// TwinCAT 3 PLC project HeatAndSteam
// ProgramVersion: 3.1.4023.0
// libraries:
//   Tc2_DataExchange, * (Beckhoff Automation GmbH)
//   Tc2_EtherCAT, * (Beckhoff Automation GmbH)
//   Tc2_MDP, * (Beckhoff Automation GmbH)
//   Tc2_ModbusSrv, * (Beckhoff Automation GmbH)
//   Tc2_Standard, * (Beckhoff Automation GmbH)
//   Tc2_SUPS, * (Beckhoff Automation GmbH)
//   Tc2_System, * (Beckhoff Automation GmbH)
//   Tc2_Utilities, * (Beckhoff Automation GmbH)
//   Tc3_DynamicMemory, * (Beckhoff Automation GmbH)
//   Tc3_EventLogger, * (Beckhoff Automation GmbH)
//   Tc3_Module, * (Beckhoff Automation GmbH)
//   Tc3_PackML_V2, * (Beckhoff Automation GmbH)
//   Tc3_PLCopen_OpcUa, * (Beckhoff Automation GmbH)
// project tree:
//   DUTs/CELLS_INFO_STRUCTURES/Development/ DUT_STRUCT_C000000_DEV.TcDUT, DUT_STRUCT_C000001_DEV.TcDUT, DUT_STRUCT_C000002_DEV.TcDUT, DUT_STRUCT_C000003_DEV.TcDUT, DUT_STRUCT_C000004_DEV.TcDUT, DUT_STRUCT_C000005_DEV.TcDUT, DUT_STRUCT_C000006_DEV.TcDUT, DUT_STRUCT_C000007_DEV.TcDUT, DUT_STRUCT_C000008_DEV.TcDUT, DUT_STRUCT_C000009_DEV.TcDUT, DUT_STRUCT_C000010_DEV.TcDUT, DUT_STRUCT_C000012_DEV.TcDUT, DUT_STRUCT_LINECONTROLLER_DEV.TcDUT, DUT_STRUCT_TRACKSERVER_DEV.TcDUT
//   DUTs/CELLS_INFO_STRUCTURES/Production/ DUT_STRUCT_C000000_PROD.TcDUT, DUT_STRUCT_C000001_PROD.TcDUT, DUT_STRUCT_C000002_PROD.TcDUT, DUT_STRUCT_C000003_PROD.TcDUT, DUT_STRUCT_C000004_PROD.TcDUT, DUT_STRUCT_C000005_PROD.TcDUT, DUT_STRUCT_C000006_PROD.TcDUT, DUT_STRUCT_C000007_PROD.TcDUT, DUT_STRUCT_C000008_PROD.TcDUT, DUT_STRUCT_C000009_PROD.TcDUT, DUT_STRUCT_C000010_PROD.TcDUT, DUT_STRUCT_C000012_PROD.TcDUT, DUT_STRUCT_LINECONTROLLER_PROD.TcDUT, DUT_STRUCT_TRACKSERVER_PROD.TcDUT
//   ECC/Basic/ADS Comm/ E_ADS_Comm_State.TcDUT (not stored), E_ADS_Comm_Type.TcDUT (not stored), FB_ADS_Comm.TcPOU (not stored)
//   ECC/Basic/Cell/ FB_Cell_Basic.TcPOU (not stored), FB_PLC_Basic.TcPOU (not stored)
//   ECC/Basic/Common Units/ E_Units.TcDUT (not stored), FB_Units.TcPOU (not stored)
//   ECC/Basic/ GVL_BASIC.TcGVL (not stored)
//   ECC/Basic/OPC Data/ E_StationJobData.TcDUT (not stored), F_NewDeviceDataX.TcPOU (not stored), ST_InputHeader.TcDUT (not stored), ST_OutputHeaderCellInformationX.TcDUT (not stored), ST_OutputHeaderMetaInformationX.TcDUT (not stored)
//   ECC/Basic/OPC Data/Sub/ E_AlarmCategory.TcDUT (not stored), E_PML_Command.TcDUT (not stored), E_PML_Mode.TcDUT (not stored), E_PML_State.TcDUT (not stored), MaterialDataX.TcDUT (not stored), MaterialXMapping.TcDUT (not stored), ST_DataPointX.TcDUT (not stored), ST_DeviceDataX.TcDUT (not stored), ST_ErrorWarningDataX.TcDUT (not stored), ST_ManipulateMLX.TcDUT (not stored), ST_MaterialDataX.TcDUT (not stored), ST_OutputHeaderCellInformationStationInformationOperationInformationX.TcDUT (not stored), ST_OutputHeaderCellInformationStationX.TcDUT (not stored), ST_OutputHeaderTransportInformationX.TcDUT (not stored), ST_SKURestriction.TcDUT (not stored), ST_ToolDataX.TcDUT (not stored), ToolDataX.TcDUT (not stored), ToolX.TcDUT (not stored), ToolXMapping.TcDUT (not stored)
//   ECC/Basic/OPC Data/Sub/Input/ ST_InputModeState.TcDUT (not stored)
//   ECC/Basic/OPC Data/Sub/Output/ ST_Energy.TcDUT (not stored), ST_Exhaust.TcDUT (not stored), ST_Fluid.TcDUT (not stored), ST_JobDataOut.TcDUT (not stored), ST_OperationalDataOPxxxxx.TcDUT (not stored), ST_OutputErrorWarning.TcDUT (not stored), ST_OutputModeState.TcDUT (not stored), ST_OutputOEE.TcDUT (not stored)
//   ECC/Basic/Station/ FB_Station_Basic.TcPOU (not stored)
//   ECC/Basic/TrackClient/DUT/ E_CellType.TcDUT (not stored), E_MMDirection.TcTLEO (not stored), E_MMStationBuffer.TcTLEO (not stored), E_MMTrafficLightColor.TcTLEO (not stored), E_MMVehicleCommand.TcTLEO (not stored), E_MMVehicleInputType.TcTLEO (not stored), ST_MethodArgumentData.TcDUT (not stored), ST_MMBuffer.TcDUT (not stored), ST_MMLocation.TcDUT (not stored), ST_MMStation.TcDUT (not stored), ST_MMVehicleFlagData.TcDUT (not stored), ST_MMVehicleStatusData.TcDUT (not stored), ST_OPCUA_MethodData.TcDUT (not stored)
//   ECC/Basic/TrackClient/Enums/ E_CarrierStatus.TcDUT (not stored), E_MMPathMotionStatus.TcTLEO (not stored), E_MMPathState.TcTLEO (not stored), E_MMServerStatus.TcTLEO (not stored), E_OPC_UA_Errors.TcDUT (not stored), E_TrackClientState.TcDUT (not stored), E_TrackState.TcDUT (not stored), E_VehicleMoveState.TcDUT (not stored)
//   ECC/Basic/TrackClient/ E_CommandDataState.TcDUT (not stored), E_MappingDataState.TcDUT (not stored), E_ReworkDataState.TcDUT (not stored), FB_TrackClient_Basic.TcPOU (not stored)
//   ECC/Basic/TrackClient/GVLs/ GlobalConstants.TcGVL (not stored)
//   ECC/Basic/TrackClient/Method Data/Cell/ ST_GetCellIndexData.TcDUT (not stored), ST_GetCellIndexDataIn.TcDUT (not stored), ST_GetCellIndexDataOut.TcDUT (not stored)
//   ECC/Basic/TrackClient/Method Data/Data/ E_MaterialType.TcDUT (not stored), E_ToolType.TcDUT (not stored), ST_AddReservationData.TcDUT (not stored), ST_AddReservationDataIn.TcDUT (not stored), ST_AddReservationDataOut.TcDUT (not stored), ST_RemoveReservationData.TcDUT (not stored), ST_RemoveReservationDataIn.TcDUT (not stored), ST_RemoveReservationDataOut.TcDUT (not stored), ST_UpdateStationBufferData.TcDUT (not stored), ST_UpdateStationBufferDataIn.TcDUT (not stored), ST_UpdateStationBufferDataOut.TcDUT (not stored), ST_UpdateVehicleDataData.TcDUT (not stored) (excluded from build), ST_UpdateVehicleDataDataIn.TcDUT (not stored) (excluded from build), ST_UpdateVehicleDataDataOut.TcDUT (not stored) (excluded from build), ST_UpdateVehicleMappingDataData.TcDUT (not stored), ST_UpdateVehicleMappingDataDataIn.TcDUT (not stored), ST_UpdateVehicleMappingDataDataOut.TcDUT (not stored), ST_UpdateVehicleMontageData.TcDUT (not stored), ST_UpdateVehicleMontageDataIn.TcDUT (not stored), ST_UpdateVehicleMontageDataOut.TcDUT (not stored), ST_UpdateVehicleOwnerData.TcDUT (not stored), ST_UpdateVehicleOwnerDataIn.TcDUT (not stored), ST_UpdateVehicleOwnerDataOut.TcDUT (not stored), ST_UpdateVehicleReservationDataData.TcDUT (not stored), ST_UpdateVehicleReservationDataDataIn.TcDUT (not stored), ST_UpdateVehicleReservationDataDataOut.TcDUT (not stored), ST_UpdateVehicleReworkDataData.TcDUT (not stored), ST_UpdateVehicleReworkDataDataIn.TcDUT (not stored), ST_UpdateVehicleReworkDataDataOut.TcDUT (not stored)
//   ECC/Basic/TrackClient/Method Data/MoveVehicle/ ST_MoveToBufferData.TcDUT (not stored), ST_MoveToBufferDataIn.TcDUT (not stored), ST_MoveToBufferDataOut.TcDUT (not stored), ST_MoveToDecisionPointData.TcDUT (not stored), ST_MoveToDecisionPointDataIn.TcDUT (not stored), ST_MoveToDecisionPointDataOut.TcDUT (not stored), ST_MoveToPositionData.TcDUT (not stored), ST_MoveToPositionDataIn.TcDUT (not stored), ST_MoveToPositionDataOut.TcDUT (not stored), ST_MoveToScannerData.TcDUT (not stored), ST_MoveToScannerDataIn.TcDUT (not stored), ST_MoveToScannerDataOut.TcDUT (not stored), ST_MoveToStationDataIn.TcDUT (not stored), ST_MoveToStationDataOut.TcDUT (not stored), ST_MoveToStationInData.TcDUT (not stored), ST_MoveToStationOutData.TcDUT (not stored), ST_MoveVehicleStatusData.TcDUT (not stored), ST_MoveVehicleStatusDataIn.TcDUT (not stored), ST_MoveVehicleStatusDataOut.TcDUT (not stored)
//   ECC/Basic/TrackClient/Method Data/Path/ ST_AddPathData.TcDUT (not stored), ST_AddPathDataIn.TcDUT (not stored), ST_AddPathDataOut.TcDUT (not stored), ST_RemovePathData.TcDUT (not stored), ST_RemovePathDataIn.TcDUT (not stored), ST_RemovePathDataOut.TcDUT (not stored), ST_ResetPathData.TcDUT (not stored), ST_ResetPathDataIn.TcDUT (not stored), ST_ResetPathDataOut.TcDUT (not stored), ST_ResumePathData.TcDUT (not stored), ST_ResumePathDataIn.TcDUT (not stored), ST_ResumePathDataOut.TcDUT (not stored), ST_StartPathData.TcDUT (not stored), ST_StartPathDataIn.TcDUT (not stored), ST_StartPathDataOut.TcDUT (not stored), ST_SuspendPathData.TcDUT (not stored), ST_SuspendPathDataIn.TcDUT (not stored), ST_SuspendPathDataOut.TcDUT (not stored)
//   ECC/Basic/TrackClient/Method Data/Segment/ ST_AddPathSegmentData.TcDUT (not stored), ST_AddPathSegmentDataIn.TcDUT (not stored), ST_AddPathSegmentDataOut.TcDUT (not stored), ST_GetPathSegmentVehicleCountData.TcDUT (not stored), ST_GetPathSegmentVehicleCountDataIn.TcDUT (not stored), ST_GetPathSegmentVehicleCountDataOut.TcDUT (not stored), ST_RemovePathSegmentData.TcDUT (not stored), ST_RemovePathSegmentDataIn.TcDUT (not stored), ST_RemovePathSegmentDataOut.TcDUT (not stored)
//   ECC/Basic/TrackClient/Method Data/Station/ ST_AddStationData.TcDUT (not stored), ST_AddStationDataIn.TcDUT (not stored), ST_AddStationDataOut.TcDUT (not stored), ST_AddStationDoubleData.TcDUT (not stored), ST_AddStationDoubleDataIn.TcDUT (not stored), ST_AddStationDoubleDataOut.TcDUT (not stored), ST_AddStationSingleData.TcDUT (not stored), ST_AddStationSingleDataIn.TcDUT (not stored), ST_AddStationSingleDataOut.TcDUT (not stored), ST_AdjustBufferPosData.TcDUT (not stored), ST_AdjustBufferPosDataIn.TcDUT (not stored), ST_AdjustBufferPosDataOut.TcDUT (not stored), ST_EnableStationData.TcDUT (not stored), ST_EnableStationDataIn.TcDUT (not stored), ST_EnableStationDataOut.TcDUT (not stored), ST_RemoveStationData.TcDUT (not stored), ST_RemoveStationDataIn.TcDUT (not stored), ST_RemoveStationDataOut.TcDUT (not stored)
//   ECC/Basic/TrackClient/Method Data/TrafficLight/ ST_AddTrafficLightData.TcDUT (not stored), ST_AddTrafficLightDataIn.TcDUT (not stored), ST_AddTrafficLightDataOut.TcDUT (not stored), ST_RemoveTrafficLightData.TcDUT (not stored), ST_RemoveTrafficLightDataIn.TcDUT (not stored), ST_RemoveTrafficLightDataOut.TcDUT (not stored), ST_SetTrafficLightColorData.TcDUT (not stored), ST_SetTrafficLightColorDataIn.TcDUT (not stored), ST_SetTrafficLightColorDataOut.TcDUT (not stored), ST_TrafficLightColorData.TcDUT (not stored), ST_TrafficLightColorDataIn.TcDUT (not stored), ST_TrafficLightColorDataOut.TcDUT (not stored)
//   ECC/Basic/TrackClient/Node Data/ E_OPC_NodeType.TcDUT (not stored), ST_ReadCellData.TcDUT (not stored), ST_ReadNodeData.TcDUT (not stored), ST_ReadPathData.TcDUT (not stored), ST_ReadPathData_OLD.TcDUT (not stored), ST_ReadStationData.TcDUT (not stored), ST_ReadVehicleData.TcDUT (not stored), ST_ReadVehicleData_OLD.TcDUT (not stored), ST_StatusCell.TcDUT (not stored), ST_StatusNode.TcDUT (not stored), ST_StatusPath.TcDUT (not stored), ST_StatusStation.TcDUT (not stored), ST_StatusVehicle.TcDUT (not stored)
//   ECC/Basic/TrackClient/Node Data/SUB/ ST_ReservationData.TcDUT (not stored)
//   ECC/Basic/TrackClient/OPC Data/ ST_InputTransport.TcDUT (not stored), ST_OutputTransport.TcDUT (not stored)
//   ECC/Basic/TrackClient/OPC Data/Sub/ ST_BufferIndexX.TcDUT (not stored), ST_CarrierX.TcDUT (not stored), ST_InputTransportAdditionalData.TcDUT (not stored), ST_InputTransportAdditionalDataMESHandShake.TcDUT (not stored), ST_InputTransportAdditionalDataSettings.TcDUT (not stored), ST_InputTransportCommand.TcDUT (not stored), ST_InputTransportConfiguration.TcDUT (not stored), ST_InputTransportMapping.TcDUT (not stored), ST_OutputTransportAdditionalData.TcDUT (not stored), ST_OutputTransportConfiguration.TcDUT (not stored), ST_OutputTransportMapping.TcDUT (not stored), ST_OutputTransportStatus.TcDUT (not stored), ST_StationBufferStatus.TcDUT (not stored), ST_StationBufferX.TcDUT (not stored), ST_StationConfigX.TcDUT (not stored), ST_StatusBuffer.TcDUT (not stored), ST_TrackLocation.TcDUT (not stored), ST_TransportMappingCarrier.TcDUT (not stored), ST_TransportMappingStationBuffer.TcDUT (not stored)
//   ECC/Cell_Unit_4/ E_VehicleOnStation.TcDUT (not stored), FB_Cell_Unit_4.TcPOU, FB_OPC_Cell_Unit_4.TcPOU (not stored), ST_VehicleInHS.TcDUT (not stored)
//   ECC/Cell_Unit_4/HeatAndSteamDeviceDriver/ FB_EMS_HS.TcPOU (not stored), U_EMS_HS_Read.TcDUT (not stored), U_EMS_HS_Write.TcDUT (not stored)
//   ECC/Cell_Unit_4/HeatAndSteamDeviceDriver/Sub/ E_EMS_HS_Status.TcDUT (not stored), ST_EMS_HS_Alarms.TcDUT (not stored), ST_EMS_HS_Command.TcDUT (not stored), ST_EMS_HS_Read.TcDUT (not stored), ST_EMS_HS_States.TcDUT (not stored), ST_EMS_HS_Write.TcDUT (not stored)
//   ECC/Cell_Unit_4/HeatAndSteam/ FB_HeatAndSteamOUT.TcPOU (not stored), F_CalcValuesHeatSteam.TcPOU (not stored), stStationVehicleCmdOut.TcDUT (not stored), E_HSStationINSeq.TcDUT (not stored), FB_HeatAndSteamIN.TcPOU (not stored)
//   ECC/Cell_Unit_4/HeatAndSteam/OPC Data/Sub/AdditionalData/ ST_InputStationHSAdditionalDataOP11600.TcDUT (not stored), ST_InputStationHSAdditionalDataOP11601.TcDUT (not stored), ST_InputStationHSAdditionalDataMESHandShake.TcDUT (not stored), ST_InputStationHSAdditionalDataSettings.TcDUT (not stored), ST_OuputStationHSAdditionalDataOP11600.TcDUT (not stored), ST_OuputStationHSAdditionalDataOP11601.TcDUT (not stored), ST_InputStationHSAdditionalData.TcDUT (not stored), ST_InputStationHSAdditionalDataGeneral.TcDUT (not stored), ST_OutputStationHSAdditionalData.TcDUT (not stored), ST_OutputStationHSAdditionalDataGeneral.TcDUT (not stored)
//   ECC/Cell_Unit_4/HeatAndSteam/OPC Data/Sub/Configuration/ ST_InputStationHSConfigurationOP11600.TcDUT (not stored), ST_InputStationHSUpcomingConfigurationOP11601.TcDUT (not stored), ST_InputStationHSConfigurationOP11601.TcDUT (not stored), ST_OutputStationHSCurrentConfigurationOP11601.TcDUT (not stored), ST_OutputStationHSUpcomingConfigurationOP11601.TcDUT (not stored), ST_InputStationHSConfiguration.TcDUT (not stored), ST_InputStationHSConfigurationGeneral.TcDUT (not stored), ST_InputStationHSUpcomingConfiguration.TcDUT (not stored), ST_InputStationHSUpcomingConfigurationOP11600.TcDUT (not stored), ST_OutputStationHSConfigurationOP11600.TcDUT (not stored), ST_OutputStationHSCurrentConfiguration.TcDUT (not stored), ST_OutputStationHSCurrentConfigurationGeneral.TcDUT (not stored), ST_OutputStationHSCurrentConfigurationOP11600.TcDUT (not stored), ST_OutputStationHSUpcomingConfiguration.TcDUT (not stored), ST_OutputStationHSUpcomingConfigurationOP11600.TcDUT (not stored)
//   ECC/Cell_Unit_4/HeatAndSteam/OPC Data/Sub/Control/ ST_InputStationHSControlOP11601.TcDUT (not stored), ST_InputStationHSControl.TcDUT (not stored), ST_InputStationHSControlGeneral.TcDUT (not stored), ST_InputStationHSControlOP11600.TcDUT (not stored)
//   ECC/Cell_Unit_4/HeatAndSteam/OPC Data/Sub/JobData/ ST_OutputStationHSJobDataOP11600.TcDUT (not stored), ST_InputStationHSJobDataOP11601.TcDUT (not stored), ST_OutputStationHSJobDataOP11601.TcDUT (not stored), ST_InputStationHSJobData.TcDUT (not stored), ST_InputStationHSJobDataOP11600.TcDUT (not stored), ST_OutputStationHSJobData.TcDUT (not stored)
//   ECC/Cell_Unit_4/HeatAndSteam/OPC Data/Sub/OperationalData/ ST_OutputStationHSOperationalDataOP11601.TcDUT (not stored), ST_OutputStationHSOperationalData.TcDUT (not stored), ST_OutputStationHSOperationalDataGeneral.TcDUT (not stored), ST_OutputStationHSOperationalDataOP11600.TcDUT (not stored)
//   ECC/Cell_Unit_4/OPC Data/ ST_Input.TcDUT (not stored), ST_Output.TcDUT (not stored)
//   ECC/Cell_Unit_4/OPC Data/Sub/ ST_InputCell.TcDUT (not stored), ST_InputCellAdditionalData.TcDUT (not stored), ST_InputCellAdditionalDataMESHandShake.TcDUT (not stored), ST_InputCellAdditionalDataSettings.TcDUT (not stored), ST_InputCellConfiguration.TcDUT (not stored), ST_InputCellConfigurationGeneral.TcDUT (not stored), ST_InputCellControl.TcDUT (not stored), ST_InputStation.TcDUT (not stored), ST_OutputCell.TcDUT (not stored), ST_OutputCellAdditionalData.TcDUT (not stored), ST_OutputCellConfiguration.TcDUT (not stored), ST_OutputCellConfigurationGeneral.TcDUT (not stored), ST_OutputCellOperationalData.TcDUT (not stored), ST_OutputCellSustainabilityData.TcDUT (not stored), ST_OutputHeader.TcDUT (not stored), ST_OutputHeaderCellInformation.TcDUT (not stored), ST_OutputHeaderCellInformationStation.TcDUT (not stored), ST_OutputHeaderCellInformationStationInformationOperationInformation.TcDUT (not stored), ST_OutputStation.TcDUT (not stored), ST_OutputCellOperationalDataGeneral.TcDUT (not stored)
//   ECC/Cell_Unit_4/HeatAndSteam/OPC Data/ ST_InputStationStationHS.TcDUT (not stored), ST_OutputStationStationHS.TcDUT (not stored)
//   ECC/Cell_Unit_4/HeatAndSteam/OPC Data/Sub/Information/ ST_OutputHeaderCellInformationStationHS.TcDUT (not stored)
//   ECC/Cell_Unit_4/HeatAndSteam/OPC Data/Sub/Sustainability/ ST_OutputStationHSSustainabilityData.TcDUT (not stored)
//   ECC/Components/ E_ComponentErrors.TcDUT (not stored), E_Cylinder_Cmd.TcDUT (not stored), E_Cylinder_Sta.TcDUT (not stored), FB_AI.TcPOU (not stored), FB_AO.TcPOU (not stored), FB_Basic.TcPOU (not stored), FB_Blink.TcPOU (not stored), FB_Cylinder.TcPOU (not stored), FB_DI.TcPOU (not stored), FB_DO.TcPOU (not stored), FB_LIN_TRAFO.TcPOU (not stored), F_ECat_OK.TcPOU (not stored), GVL_Components.TcGVL (not stored)
//   ECC/Components/TwinSAFE/ E_TwinSAFE_Group_Diag.TcDUT (not stored), E_TwinSAFE_Group_State.TcDUT (not stored), E_TwinSAFE_Logic_State.TcDUT (not stored), FB_TwinSAFE_Group.TcPOU (not stored)
//   ECC/Tools/ E_Method.TcDUT (not stored), E_OPCUA_Client_Seq.TcDUT (not stored), FB_CheckHeartBeat.TcPOU (not stored), FB_GenerateHeartBeat.TcPOU (not stored), FB_GetCPULoad.TcPOU (not stored), FB_GetCPULoadPLC.TcPOU (not stored), FB_GetCPUTemp.TcPOU (not stored), FB_GetIPCSerial.TcPOU (not stored), FB_GetSafetyTemp.TcPOU (not stored), FB_GetTimePML.TcPOU (not stored), FB_OPCUA_Client_Basic.TcPOU (not stored), FB_OPCUA_Client_CallMethod.TcPOU (not stored), FB_OPCUA_Client_ReadVar.TcPOU (not stored), FB_OPCUA_GetRecipe.TcPOU (not stored), FB_OPCUA_ReadVar_BAK.TcPOU (not stored), F_Array_Sort.TcPOU (not stored), F_LogLine.TcPOU (not stored), F_StringCompNoCase.TcPOU (not stored), ST_OPC_Client_Data.TcDUT (not stored), ST_OutputArgInfoAndData_Basis.TcDUT (not stored), ST_Test.TcDUT (not stored)
//   ECC/Tools/LogToFile/ FB_GetFifo.TcPOU (not stored), FB_LogToFile.TcPOU (not stored), FB_SetFifo.TcPOU (not stored), F_LogFile.TcPOU (not stored), F_PadWith.TcPOU (not stored), GVL_Log.TcGVL (not stored), ST_String_FIFO.TcDUT (not stored)
//   ECC/TrackClient/Buffer Control/ FB_BufferControl.TcPOU (not stored), ST_BufferControl.TcDUT (not stored)
//   ECC/TrackClient/Enums/ E_BufferState.TcDUT (not stored), E_BufferStates.TcDUT (not stored), E_PostBufferInState.TcDUT (not stored), E_DecisionPointState.TcDUT (not stored), E_ExitPointState.TcDUT (not stored), E_StationState.TcDUT (not stored), E_PostBufferOutState.TcDUT (not stored)
//   ECC/TrackClient/ FB_TrackClient.TcPOU (not stored)
//   ECC/TrackClient/Station Control/ E_StationBufferState.TcDUT (not stored), E_StationInOutState.TcDUT (not stored), FB_StationControl.TcPOU (not stored), ST_StationControlData.TcDUT (not stored)
//   GVLs/ GVL.TcGVL
//   / PlcTask.TcTTO (not stored)
//   POUs/ MAIN.TcPOU
// real-time tasks:
//   TASK PlcTask: cycle T#10ms, priority 20, ADS port 350
// I/O:
//   DEVICE PCI (EtherCAT) (disabled), AmsNetId 10.128.16.81.2.1
//     BusCoupler (EK1200) [EK1200-5000 EtherCAT Power supply (2A E-Bus)]
//       License (EL6070-0033) [EL6070-0033 1Ch. Licence key terminal, individual licences]
//       End (EL9011) [EL9011 End Terminal]
// variable links:
//   HeatAndSteam/HeatAndSteam Instance <-> PCI (EtherCAT)/BusCoupler (EK1200)/License (EL6070-0033)
//     PlcTask Inputs/MAIN.fbUnit4.License_AdsAdrr <-> InfoData/AdsAddr
//     PlcTask Inputs/MAIN.fbUnit4.License_State <-> InfoData/State
//     PlcTask Inputs/MAIN.fbUnit4.fbSafetyTemp.sSafetyNetID/port <-> InfoData/AdsAddr/port

// ---- DUTs/CELLS_INFO_STRUCTURES/Development/DUT_STRUCT_C000000_DEV.TcDUT
TYPE DUT_STRUCT_C000000_DEV :
STRUCT
	sCellName			:STRING := 'C000000';
	sIpAddress			:STRING := '10.155.180.5';
	sAmsNetId			:STRING := '10.155.180.5.1.1';
	sOpcUaURL			:STRING := 'opc.tcp://10.155.180.5:4840';
	sUhfRfidOpcUaURL	:STRING := 'opc.tcp://10.155.180.5:4840';
	sHfRfidOpcUaURL		:STRING := 'opc.tcp://10.155.180.5:4840';
	sStation1			:STRING := 'S00000A';
END_STRUCT
END_TYPE

// ---- DUTs/CELLS_INFO_STRUCTURES/Development/DUT_STRUCT_C000001_DEV.TcDUT
TYPE DUT_STRUCT_C000001_DEV :
STRUCT
	sCellName			:STRING := 'C000001';
	sIpAddress			:STRING := '';
	sAmsNetId			:STRING := '';
	sOpcUaURL			:STRING := 'opc.tcp://:4840';
	sStation1			:STRING := 'S000008';
	sStation2			:STRING := 'S000009';
END_STRUCT
END_TYPE

// ---- DUTs/CELLS_INFO_STRUCTURES/Development/DUT_STRUCT_C000002_DEV.TcDUT
TYPE DUT_STRUCT_C000002_DEV :
STRUCT
	sCellName			:STRING := 'C000002';
	sIpAddress			:STRING := '';
	sAmsNetId			:STRING := '';
	sOpcUaURL			:STRING := 'opc.tcp://:4840';
	sStation1			:STRING := 'S000007';
END_STRUCT
END_TYPE

// ---- DUTs/CELLS_INFO_STRUCTURES/Development/DUT_STRUCT_C000003_DEV.TcDUT
TYPE DUT_STRUCT_C000003_DEV :
STRUCT
	sCellName			:STRING := 'C000003';
	sIpAddress			:STRING := '';
	sAmsNetId			:STRING := '';
	sOpcUaURL			:STRING := 'opc.tcp://:4840';
	sStation1			:STRING := 'S000006';
END_STRUCT
END_TYPE

// ---- DUTs/CELLS_INFO_STRUCTURES/Development/DUT_STRUCT_C000004_DEV.TcDUT
TYPE DUT_STRUCT_C000004_DEV :
STRUCT
	sCellName			:STRING := 'C000004';
	sIpAddress			:STRING := '10.155.180.12';
	sAmsNetId			:STRING := '10.155.180.12.1.1';
	sOpcUaURL			:STRING := 'opc.tcp://10.155.180.12:4840';
	sStation1			:STRING := 'S000003';
END_STRUCT
END_TYPE

// ---- DUTs/CELLS_INFO_STRUCTURES/Development/DUT_STRUCT_C000005_DEV.TcDUT
TYPE DUT_STRUCT_C000005_DEV :
STRUCT
	sCellName			:STRING := 'C000005';
	sIpAddress			:STRING := '';
	sAmsNetId			:STRING := '';
	sOpcUaURL			:STRING := 'opc.tcp://:4840';
	sStation1			:STRING := 'S000001';
END_STRUCT
END_TYPE

// ---- DUTs/CELLS_INFO_STRUCTURES/Development/DUT_STRUCT_C000006_DEV.TcDUT
TYPE DUT_STRUCT_C000006_DEV :
STRUCT
	sCellName			:STRING := 'C000006';
	sIpAddress			:STRING := '';
	sAmsNetId			:STRING := '';
	sOpcUaURL			:STRING := 'opc.tcp://:4840';
	sStation1			:STRING := 'S000002';
END_STRUCT
END_TYPE

// ---- DUTs/CELLS_INFO_STRUCTURES/Development/DUT_STRUCT_C000007_DEV.TcDUT
TYPE DUT_STRUCT_C000007_DEV :
STRUCT
	sCellName			:STRING := 'C0000007';
	sIpAddress			:STRING := '';
	sAmsNetId			:STRING := '';
	sOpcUaURL			:STRING := 'opc.tcp://:4840';
	sStation1			:STRING := 'S00000B';
END_STRUCT
END_TYPE

// ---- DUTs/CELLS_INFO_STRUCTURES/Development/DUT_STRUCT_C000008_DEV.TcDUT
TYPE DUT_STRUCT_C000008_DEV :
STRUCT
	sCellName			:STRING := 'C000008';
	sIpAddress			:STRING := '';
	sAmsNetId			:STRING := '';
	sOpcUaURL			:STRING := 'opc.tcp://:4840';
	sStation1			:STRING := 'S000005';
END_STRUCT
END_TYPE

// ---- DUTs/CELLS_INFO_STRUCTURES/Development/DUT_STRUCT_C000009_DEV.TcDUT
TYPE DUT_STRUCT_C000009_DEV :
STRUCT
	sCellName			:STRING := 'C000009';
	sIpAddress			:STRING := '';
	sAmsNetId			:STRING := '';
	sOpcUaURL			:STRING := 'opc.tcp://:4840';
	sUhfRfidOpcUaURL	:STRING := 'opc.tcp://:4840';
	sHfRfidOpcUaURL		:STRING := 'server:opc.tcp://:4840';
	sStation1			:STRING := 'S000004';
	sLastingPC			:STRING := '';
END_STRUCT
END_TYPE

// ---- DUTs/CELLS_INFO_STRUCTURES/Development/DUT_STRUCT_C000010_DEV.TcDUT
TYPE DUT_STRUCT_C000010_DEV :
STRUCT
	sCellName			:STRING := 'C000010';
	sIpAddress			:STRING := '';
	sAmsNetId			:STRING := '';
	sOpcUaURL			:STRING := 'opc.tcp://:4840';
	sStation1			:STRING := 'S00005D';
	sStation2			:STRING := 'S00005A';
END_STRUCT
END_TYPE

// ---- DUTs/CELLS_INFO_STRUCTURES/Development/DUT_STRUCT_C000012_DEV.TcDUT
TYPE DUT_STRUCT_C000012_DEV :
STRUCT
	sCellName			:STRING := 'C000012';
	sIpAddress			:STRING := '';
	sAmsNetId			:STRING := '';
	sOpcUaURL			:STRING := 'opc.tcp://:4840';
	sStation1			:STRING := 'S000010';
END_STRUCT
END_TYPE

// ---- DUTs/CELLS_INFO_STRUCTURES/Development/DUT_STRUCT_LINECONTROLLER_DEV.TcDUT
TYPE DUT_STRUCT_LINECONTROLLER_DEV :
STRUCT
	sCellName			:STRING := 'LINECONTROLLER';
	sIpAddress			:STRING := '10.155.180.8';
	sAmsNetId			:STRING := '';
END_STRUCT
END_TYPE

// ---- DUTs/CELLS_INFO_STRUCTURES/Development/DUT_STRUCT_TRACKSERVER_DEV.TcDUT
TYPE DUT_STRUCT_TRACKSERVER_DEV :
STRUCT
	sCellName			:STRING := 'TRACKSERVER';
	sIpAddress			:STRING := '10.155.180.10';
	sAmsNetId			:STRING := '10.155.180.10.1.1';
END_STRUCT
END_TYPE

// ---- DUTs/CELLS_INFO_STRUCTURES/Production/DUT_STRUCT_C000000_PROD.TcDUT
TYPE DUT_STRUCT_C000000_PROD :
STRUCT
	sCellName			:STRING := 'C000000';
	sIpAddress			:STRING := '10.38.190.130';
	sAmsNetId			:STRING := '10.38.190.130.1.1';
	sOpcUaURL			:STRING := 'opc.tcp://10.38.190.130:4840';
	sUhfRfidOpcUaURL	:STRING := 'opc.tcp://10.38.190.132:4840';
	sHfRfidOpcUaURL		:STRING := 'opc.tcp://10.38.190.134:4840';
	sStation1			:STRING := 'S00000A';
END_STRUCT
END_TYPE

// ---- DUTs/CELLS_INFO_STRUCTURES/Production/DUT_STRUCT_C000001_PROD.TcDUT
TYPE DUT_STRUCT_C000001_PROD :
STRUCT
	sCellName			:STRING := 'C000001';
	sIpAddress			:STRING := '10.38.191.0';
	sAmsNetId			:STRING := '10.38.191.0.1.1';
	sOpcUaURL			:STRING := 'opc.tcp://10.38.191.0:4840';
	sStation1			:STRING := 'S000008';
	sStation2			:STRING := 'S000009';
END_STRUCT
END_TYPE

// ---- DUTs/CELLS_INFO_STRUCTURES/Production/DUT_STRUCT_C000002_PROD.TcDUT
TYPE DUT_STRUCT_C000002_PROD :
STRUCT
	sCellName			:STRING := 'C000002';
	sIpAddress			:STRING := '10.38.191.20';
	sAmsNetId			:STRING := '10.38.191.20.1.1';
	sOpcUaURL			:STRING := 'opc.tcp://10.38.191.20:4840';
	sStation1			:STRING := 'S000007';
END_STRUCT
END_TYPE

// ---- DUTs/CELLS_INFO_STRUCTURES/Production/DUT_STRUCT_C000003_PROD.TcDUT
TYPE DUT_STRUCT_C000003_PROD :
STRUCT
	sCellName			:STRING := 'C000003';
	sIpAddress			:STRING := '10.38.191.40';
	sAmsNetId			:STRING := '10.38.191.40.1.1';
	sOpcUaURL			:STRING := 'opc.tcp://10.38.191.40:4840';
	sStation1			:STRING := 'S000006';
END_STRUCT
END_TYPE

// ---- DUTs/CELLS_INFO_STRUCTURES/Production/DUT_STRUCT_C000004_PROD.TcDUT
TYPE DUT_STRUCT_C000004_PROD :
STRUCT
	sCellName			:STRING := 'C000004';
	sIpAddress			:STRING := '10.38.190.201';
	sAmsNetId			:STRING := '10.38.190.201.1.1';
	sOpcUaURL			:STRING := 'opc.tcp://10.38.190.201:4840';
	sStation1			:STRING := 'S000003';
END_STRUCT
END_TYPE

// ---- DUTs/CELLS_INFO_STRUCTURES/Production/DUT_STRUCT_C000005_PROD.TcDUT
TYPE DUT_STRUCT_C000005_PROD :
STRUCT
	sCellName			:STRING := 'C000005';
	sIpAddress			:STRING := '10.38.190.204';
	sAmsNetId			:STRING := '10.38.190.204.1.1';
	sOpcUaURL			:STRING := 'opc.tcp://10.38.190.204:4840';
	sStation1			:STRING := 'S000001';
END_STRUCT
END_TYPE

// ---- DUTs/CELLS_INFO_STRUCTURES/Production/DUT_STRUCT_C000006_PROD.TcDUT
TYPE DUT_STRUCT_C000006_PROD :
STRUCT
	sCellName			:STRING := 'C000006';
	sIpAddress			:STRING := '10.38.190.200';
	sAmsNetId			:STRING := '10.38.190.200.1.1';
	sOpcUaURL			:STRING := 'opc.tcp://10.38.190.200:4840';
	sStation1			:STRING := 'S000002';
END_STRUCT
END_TYPE

// ---- DUTs/CELLS_INFO_STRUCTURES/Production/DUT_STRUCT_C000007_PROD.TcDUT
TYPE DUT_STRUCT_C000007_PROD :
STRUCT
	sCellName			:STRING := 'C0000007';
	sIpAddress			:STRING := '10.38.190.203';
	sAmsNetId			:STRING := '10.38.190.203.1.1';
	sOpcUaURL			:STRING := 'opc.tcp://10.38.190.203:4840';
	sStation1			:STRING := 'S00000B';
END_STRUCT
END_TYPE

// ---- DUTs/CELLS_INFO_STRUCTURES/Production/DUT_STRUCT_C000008_PROD.TcDUT
TYPE DUT_STRUCT_C000008_PROD :
STRUCT
	sCellName			:STRING := 'C000008';
	sIpAddress			:STRING := '10.38.190.202';
	sAmsNetId			:STRING := '10.38.190.202.1.1';
	sOpcUaURL			:STRING := 'opc.tcp://10.38.190.202:4840';
	sStation1			:STRING := 'S000005';
END_STRUCT
END_TYPE

// ---- DUTs/CELLS_INFO_STRUCTURES/Production/DUT_STRUCT_C000009_PROD.TcDUT
TYPE DUT_STRUCT_C000009_PROD :
STRUCT
	sCellName			:STRING := 'C000009';
	sIpAddress			:STRING := '10.38.191.60';
	sAmsNetId			:STRING := '10.38.191.60.1.1';
	sOpcUaURL			:STRING := 'opc.tcp://10.38.191.60:4840';
	sUhfRfidOpcUaURL	:STRING := 'opc.tcp://10.38.190.132:4840';
	sHfRfidOpcUaURL		:STRING := 'server:opc.tcp://10.38.191.66:4840';
	sStation1			:STRING := 'S000004';
	sLastingPC			:STRING := '10.38.191.65';
END_STRUCT
END_TYPE

// ---- DUTs/CELLS_INFO_STRUCTURES/Production/DUT_STRUCT_C000010_PROD.TcDUT
TYPE DUT_STRUCT_C000010_PROD :
STRUCT
	sCellName			:STRING := 'C000010';
	sIpAddress			:STRING := '10.38.191.100';
	sAmsNetId			:STRING := '10.38.191.100.1.1';
	sOpcUaURL			:STRING := 'opc.tcp://10.38.191.100:4840';
	sStation1			:STRING := 'S00005D';
	sStation2			:STRING := 'S00005A';
END_STRUCT
END_TYPE

// ---- DUTs/CELLS_INFO_STRUCTURES/Production/DUT_STRUCT_C000012_PROD.TcDUT
TYPE DUT_STRUCT_C000012_PROD :
STRUCT
	sCellName			:STRING := 'C000012';
	sIpAddress			:STRING := '10.38.191.140';
	sAmsNetId			:STRING := '10.38.191.140.1.1';
	sOpcUaURL			:STRING := 'opc.tcp://10.38.191.140:4840';
	sStation1			:STRING := 'S000010';
END_STRUCT
END_TYPE

// ---- DUTs/CELLS_INFO_STRUCTURES/Production/DUT_STRUCT_LINECONTROLLER_PROD.TcDUT
TYPE DUT_STRUCT_LINECONTROLLER_PROD :
STRUCT
	sCellName			:STRING := 'LINECONTROLLER';
	sIpAddress			:STRING := '10.38.190.120';
	sAmsNetId			:STRING := '';
END_STRUCT
END_TYPE

// ---- DUTs/CELLS_INFO_STRUCTURES/Production/DUT_STRUCT_TRACKSERVER_PROD.TcDUT
TYPE DUT_STRUCT_TRACKSERVER_PROD :
STRUCT
	sCellName			:STRING := 'TRACKSERVER';
	sIpAddress			:STRING := '10.38.190.121';
	sAmsNetId			:STRING := '10.38.190.121.1.1';
END_STRUCT
END_TYPE

// ---- GVLs/GVL.TcGVL
VAR_GLOBAL CONSTANT
	{attribute 'OPC.UA.DA':='1'}
	{attribute 'OPC.UA.DA.Access' := '1'}
	{attribute 'OPC.UA.DA.Description' := 'SW Version'}
	sSWVersion			: STRING := '0.1';

	iNoOfRecipeData		: UINT := 100;
END_VAR
VAR_GLOBAL
	bLogToOutputWindow	: BOOL;		// if TRUE it will log all logs to file AND to output window
	
	// cells info for PRODUCTION
	C000000_PROD				:DUT_STRUCT_C000000_PROD;
	C000001_PROD				:DUT_STRUCT_C000001_PROD;
	C000002_PROD				:DUT_STRUCT_C000002_PROD;
	C000003_PROD				:DUT_STRUCT_C000003_PROD;
	C000004_PROD				:DUT_STRUCT_C000004_PROD;
	C000005_PROD				:DUT_STRUCT_C000005_PROD;
	C000006_PROD				:DUT_STRUCT_C000006_PROD;
	C000007_PROD				:DUT_STRUCT_C000007_PROD;
	C000008_PROD				:DUT_STRUCT_C000008_PROD;
	C000009_PROD				:DUT_STRUCT_C000009_PROD;
	C000010_PROD				:DUT_STRUCT_C000010_PROD;
	C000012_PROD				:DUT_STRUCT_C000012_PROD;
	TrackServer_PROD			:DUT_STRUCT_TRACKSERVER_PROD;
	LineController_PROD			:DUT_STRUCT_LINECONTROLLER_PROD;
	
	// cells info for DEVELOPMENT
	C000000_DEV					:DUT_STRUCT_C000000_DEV;
	C000001_DEV					:DUT_STRUCT_C000001_DEV;
	C000002_DEV					:DUT_STRUCT_C000002_DEV;
	C000003_DEV					:DUT_STRUCT_C000003_DEV;
	C000004_DEV					:DUT_STRUCT_C000004_DEV;
	C000005_DEV					:DUT_STRUCT_C000005_DEV;
	C000006_DEV					:DUT_STRUCT_C000006_DEV;
	C000007_DEV					:DUT_STRUCT_C000007_DEV;
	C000008_DEV					:DUT_STRUCT_C000008_DEV;
	C000009_DEV					:DUT_STRUCT_C000009_DEV;
	C000010_DEV					:DUT_STRUCT_C000010_DEV;
	C000012_DEV					:DUT_STRUCT_C000012_DEV;
	TrackServer_DEV				:DUT_STRUCT_TRACKSERVER_DEV;
	LineController_DEV			:DUT_STRUCT_LINECONTROLLER_DEV;
END_VAR

// ---- ECC/Cell_Unit_4/FB_Cell_Unit_4.TcPOU
FUNCTION_BLOCK FB_Cell_Unit_4 EXTENDS FB_Cell_Basic
VAR_INPUT
END_VAR
VAR_OUTPUT
	bError						: BOOL;
	iErrorID					: BOOL;
END_VAR
VAR_IN_OUT
	// Bridge data
	Input						: ST_Input;
	Output						: ST_Output;
END_VAR
VAR
// Local vars
	eSeq						: E_VehicleOnStation;
	tonSeqTimer					: TON;
	aVehiclesStationFIFO		: ARRAY[1..10] OF ST_VehicleInHS;
	aDummyVehicleStationData	: ST_VehicleInHS;
	fDistanceStation2Station	: REAL; //Distance between stations

	stDeviceInfo				: ST_DeviceIdentification;			// Device information such as serial no.
	stVehicleDataOnStation		: ST_ReadVehicleData;
	nPLCVersion					: UINT:=0;
	nScannerInterfaceVersion	: UINT:=0;	
	bInitDone					: BOOL;
	bVehicleEnterStationOS	 	: BOOL;
	bVehicleMoveToStation		: BOOL;
	iRes						: INT;
	diFifoLogTimer				: UINT;
	diVehiclesInDevice			: UINT;
	
	tonVehicleDataRead			: TON;	// To trig reading of data for vehicles in the FIFO buffer

// FunctionBlocks:
	fbStationINHeatAndSteam		: FB_HeatAndSteamIN;
	fbStationOUTHeatAndSteam	: FB_HeatAndSteamOUT;
	fbTrack						: FB_TrackClient;
	
// Start op procedure
	bBypassTrack	:	BOOL;
	nCheckValid		:	UINT;
	nIndx			:	UINT;
	nIndxStart		:	UINT;
	nIndxDone		:	UINT;
	fVel			:	REAL;
	fAcc			:	REAL;
	bStartupPrd		:	BOOL;
	
// Error / Warnings
	iST1ErrWarDataChange	: UINT;
	iST2ErrWarDataChange	: UINT;
	iTCErrWarDataChange		: UINT;
END_VAR

SUPER^(	stModeStateIn := Input.Cell.ModeState,
		stModeStateOut := Output.Cell.ModeState,
		stOEE := Output.Cell.OEE,
		stErrorWarning := Output.Cell.ErrorWarning);

// Init FB's
M_Init();

// Run components
M_Components();
		
// Device controller
M_Device_Sequence();

// Error and warnings
M_ErrorWarning();

//Sustainability Data
M_SustainabilityDataHandling();

//Clear all ticket data
IF Input.Cell.AdditionalData.ClearAll THEN
	Input.Cell.AdditionalData.ClearAll R= M_ClearAll();
END_IF

// Update PackML state/modes variables from local values
bEStopOK := TRUE;
bStartLocal;
bStopLocal;
bClearLocal;
bResetLocal := ((eCurrentState = E_PMLState.ePMLState_Complete) AND (eCommand = E_PMLCommand.ePMLCommand_Undefined)); // Automatic back to Idle when finished
bHoldLocal;
bProductionLocal;
bManualLocal;

{attribute 'object_name' := 'M_Aborted'}
METHOD M_Aborted
END_METHOD

{attribute 'object_name' := 'M_Aborting'}
METHOD M_Aborting
// Stop all moving parts


// Abort is handled internally in Brushing Station FB, follows Cell unit state!
//IF (fbScanner1.stModeStateOut.CurrentMode = E_PML_State.Aborted) THEN
//	M_StateComplete();	
//END_IF


// No moving parts, go straight to nest state
//eCommand := E_PML_Command.Undefined;
M_StateComplete();
END_METHOD

METHOD PROTECTED M_CarrierFinishInfeedToTrack : BOOL
VAR_INPUT
END_VAR

// TODO!!!
M_CarrierFinishInfeedToTrack := TRUE;
END_METHOD

METHOD PROTECTED M_CarrierFinishOutfeedToTrack : BOOL
VAR_INPUT
END_VAR

// TODO!!!
M_CarrierFinishOutfeedToTrack := TRUE;
END_METHOD

METHOD PROTECTED M_CarrierReadyInfeedFromTrack : BOOL
VAR_INPUT
END_VAR

// TODO!!!
M_CarrierReadyInfeedFromTrack := FALSE;
END_METHOD

METHOD PROTECTED M_CarrierReadyOutfeedFromTrack : BOOL
VAR_INPUT
END_VAR

// TODO!!!
M_CarrierReadyOutfeedFromTrack := TRUE;
END_METHOD

METHOD M_ClearAll : BOOL
VAR_INPUT
END_VAR
VAR
	i : USINT;
END_VAR
//Clear all ticket data on cell from OPC command

//Clear Station(s) and TrackClient
IF fbStationINHeatAndSteam.M_ClearAll() AND fbStationOUTHeatAndSteam.M_ClearAll() THEN
	M_ClearAll := fbTrack.M_ClearAll();
END_IF
	
//Clear Cell
IF M_ClearAll THEN
	 eSeq := E_VehicleOnStation.Idle;
	 
	 //Clean out FIFO
	FOR i := 1 TO 9 DO
		aVehiclesStationFIFO[i] := aDummyVehicleStationData;
	END_FOR	
	F_Logfile('Cell - All data cleared!');
END_IF
END_METHOD

{attribute 'object_name' := 'M_Clearing'}
METHOD M_Clearing
// Reset safety system

//fbScanner1.nCellStateCmd := E_PML_Command.Clear;

//fbTrack.bReset := TRUE;

//IF ((fbScanner1.stModeStateOut.CurrentMode = E_PML_State.idle) OR (fbScanner1.stModeStateOut.CurrentMode = E_PML_State.stopped)) THEN
//	M_StateComplete();
	
//	fbTrack.bReset := FALSE;
//END_IF
//eCommand := E_PML_Command.Undefined;
M_StateComplete();
END_METHOD

{attribute 'object_name' := 'M_Complete'}
METHOD M_Complete
END_METHOD

{attribute 'object_name' := 'M_Completing'}
METHOD M_Completing

VAR
	sLowHighUpperID : STRING;	
	iRes			: INT;
END_VAR

//eCommand := E_PML_Command.Undefined;
M_StateComplete();
END_METHOD

METHOD PROTECTED M_Components : BOOL
VAR_INPUT
END_VAR
VAR
END_VAR
// Run component blocks
END_METHOD

METHOD M_Device_Sequence
VAR_INPUT
END_VAR
VAR
	i			: UINT;
	iRes		: INT;
	bMoveToNext	: BOOL;
END_VAR
// Heart beat
iHeartBeatFromMES := Input.Header.HeartBeat;
Output.Header.HeartBeat := iHeartBeatToMES;

// Run Station(s) (define when each needs to run)
fbStationINHeatAndSteam(
	aVehiclesStationFIFO:= aVehiclesStationFIFO,
	stReservation:= fbTrack.P_stReservation,
	stModeStateIn:= Input.Station.Station1.ModeState, 
	stModeStateOut := Output.Station.Station1.ModeState,
	bVehicleReadyAtInput:= eSeq <> E_VehicleOnStation.Idle, 
	bVehicleReadyAtOutput:= , 
	nCellStateCmd:= DINT_TO_UINT(eCommand),
	stJobDataIn:= Input.Station.Station1.JobData,  
	stConfigIn:= Input.Station.Station1.CurrentConfiguration, 
	stUpcomingConfigIn:= Input.Station.Station1.UpcomingConfiguration, 
	stControlIn := Input.Station.Station1.Control,
	stAdditionalDataIn := Input.Station.Station1.AdditionalData,
	sDistanceInDevice := Input.Transport.Configuration.Stations[2].StationLocation1.Position - Input.Transport.Configuration.Stations[1].StationLocation1.Position,
	stVehicleDataStaion := fbTrack.P_stVehicleDataOnStation,
	stJobDataOut := Output.Station.Station1.JobData,  
	stOEE := Output.Station.Station1.OEE, 
	stErrorWarning := Output.Station.Station1.ErrorWarning, 
	stConfigOut := Output.Station.Station1.CurrentConfiguration,
	stUpcomingConfigOut := Output.Station.Station1.UpcomingConfiguration,
	stOperationalDataOut := Output.Station.Station1.OperationalData, 
	stSustainabilityData := Output.Station.Station1.SustainabilityData, 
	stAdditionalDataOut := Output.Station.Station1.AdditionalData 	);
	
fbStationOUTHeatAndSteam(
	stModeStateIn:= Input.Station.Station2.ModeState, 
	stModeStateOut := Output.Station.Station2.ModeState,
	bVehicleReadyAtInput:= , 
	bVehicleReadyAtOutput:= , 
	nCellStateCmd:= DINT_TO_UINT(eCommand),
	stJobDataIn:= Input.Station.Station2.JobData,  
	stConfigIn:= Input.Station.Station2.CurrentConfiguration, 
	stUpcomingConfigIn:= Input.Station.Station2.UpcomingConfiguration, 
	stControlIn := Input.Station.Station2.Control,
	stAdditionalDataIn := Input.Station.Station1.AdditionalData,
	stJobDataOut := Output.Station.Station2.JobData,  
	stOEE := Output.Station.Station2.OEE, 
	stErrorWarning := Output.Station.Station2.ErrorWarning, 
	stConfigOut := Output.Station.Station2.CurrentConfiguration,
	stUpcomingConfigOut := Output.Station.Station2.UpcomingConfiguration,
	stOperationalDataOut := Output.Station.Station2.OperationalData, 
	stSustainabilityData := Output.Station.Station2.SustainabilityData, 
	stAdditionalDataOut := Output.Station.Station2.AdditionalData 	);

	
// Run Track Client
fbTrack(bEnable := , // Enabled in State Resetting
		bEStopOK := TRUE,
		bSuspend := , 
		bReset:= , 
		stCommand:= Input.Transport.Command,
		stMappingIn:= input.Transport.Mapping,
		stAdditionalDataIn:= Input.Transport.AdditionalData,
		bConnectedMethod=> , 
		bBusyMethod=> , 
		bConnectedNode=> , 
		bErrorMethod=> , 
		nErrorMethodID=> , 
		bErrorNode=> , 
		nErrorNodeID=> , 
		stStatus := Output.Transport.Status,
		stMappingOut := Output.Transport.Mapping, 
		stAdditionaldataOut := Output.Transport.AdditionalData,
		bStarted=> , 
		bSuspended=> 	);


//Set Station ready for vehicle to track
fbTrack.P_StationEmptyReady := eSeq = E_VehicleOnStation.Idle;
//fbTrack.P_bStationReady:=fbStationINHeatAndSteam.bStationReadyIn;

//Vehicles on station FIFO handling
M_VehicleOnStation(iCarrierCount=>diVehiclesInDevice);


//Set station empty for track - for vehicles going straight through
fbTrack.P_bStationEmpty:= diVehiclesInDevice = 0;

//Set FIFO for Station IN and Track Client
//fbStationINHeatAndSteam.P_CarriersFIFO := aVehiclesStationFIFO;
fbTrack.P_CarriersFIFO := aVehiclesStationFIFO;
END_METHOD

METHOD PROTECTED M_ErrorWarning
VAR_INPUT
END_VAR
VAR
	iAlNo				: UINT;
	iNoOfAlarms			: UINT;
	iNoOfWarnings		: UINT;
	bST1ErrWarDataChange: BOOL;
	bST2ErrWarDataChange: BOOL;
	bCellDataChange		: BOOL;
	bTCErrWarDataChange	: BOOL;
END_VAR
//Alarm / Warnings Cell
//bCellDataChange S= 
//M_ErrorWarningObj(arErrorWaringData:= arErrorWarningDataCell,
//	bActive:= eLineCtrl_EStop <> E_TwinSAFE_Logic_State.RUN, 
//	iErrorWarningType:= 2, 
//	diErrorWarningID:= E_AlarmCategory.Safety + 0, 
//	sDeviceID:= 'Global Safety',
//	iSeverity:= 2, 
//	iNativeID:= 0, 
//	sNativeMessage:= 'Emergency stop Line Controller');

//bCellDataChange S= 
//M_ErrorWarningObj(arErrorWaringData:= arErrorWarningDataCell,
//	bActive:= NOT bEStop_OK, 
//	iErrorWarningType:= 2, 
//	diErrorWarningID:= E_AlarmCategory.Safety + 20, 
//	sDeviceID:= 'Local Safety',
//	iSeverity:= 2, 
//	iNativeID:= 0, 
//	sNativeMessage:= 'Emergency stop Cell');

//bCellDataChange S= 
//M_ErrorWarningObj(arErrorWaringData:= arErrorWarningDataCell,
//	bActive:= eSHL_F70 <> E_TwinSAFE_Logic_State.RUN, 
//	iErrorWarningType:= 2, 
//	diErrorWarningID:= E_AlarmCategory.Safety + 21, 
//	sDeviceID:= 'Local Safety',
//	iSeverity:= 2, 
//	iNativeID:= 0, 
//	sNativeMessage:= 'Emergency stop Robot');
	
//bCellDataChange S= 
//M_ErrorWarningObj(arErrorWaringData:= arErrorWarningDataCell,
//	bActive:= NOT bDoor_OK, 
//	iErrorWarningType:= 2, 
//	diErrorWarningID:= E_AlarmCategory.Safety + 22, 
//	sDeviceID:= 'Local Safety',
//	iSeverity:= 2, 
//	iNativeID:= 0, 
//	sNativeMessage:= 'Cell Door 1 Not OK');
	
//bCellDataChange S= 
//M_ErrorWarningObj(arErrorWaringData:= arErrorWarningDataCell,
//	bActive:= stStatusData.e03_11_AK01_M3011 = E_Cylinder_Sta.Cyl_Sta_Err, 
//	iErrorWarningType:= 2, 
//	diErrorWarningID:= E_AlarmCategory.LifterStation1Device + 0, 
//	sDeviceID:= 'Lifter Station 1',
//	iSeverity:= 2, 
//	iNativeID:= 0, 
//	sNativeMessage:= 'Error Radial Gripper');
	
//bCellDataChange S= 
//M_ErrorWarningObj(arErrorWaringData:= arErrorWarningDataCell,
//	bActive:= stStatusData.e03_11_AK01_M3015 = E_Cylinder_Sta.Cyl_Sta_Err, 
//	iErrorWarningType:= 2, 
//	diErrorWarningID:= E_AlarmCategory.LifterStation1Device + 1, 
//	sDeviceID:= 'Lifter Station 1',
//	iSeverity:= 2, 
//	iNativeID:= 0, 
//	sNativeMessage:= 'Error Lifter Cylinder');
	
//bCellDataChange S= 
//M_ErrorWarningObj(arErrorWaringData:= arErrorWarningDataCell,
//	bActive:= stStatusData.e03_11_AK01_M3111 = E_Cylinder_Sta.Cyl_Sta_Err, 
//	iErrorWarningType:= 2, 
//	diErrorWarningID:= E_AlarmCategory.LifterStation2Device + 0, 
//	sDeviceID:= 'Lifter Station 2',
//	iSeverity:= 2, 
//	iNativeID:= 0, 
//	sNativeMessage:= 'Error Radial Gripper');
	
//bCellDataChange S= 
//M_ErrorWarningObj(arErrorWaringData:= arErrorWarningDataCell,
//	bActive:= stStatusData.e03_11_AK01_M3115 = E_Cylinder_Sta.Cyl_Sta_Err, 
//	iErrorWarningType:= 2, 
//	diErrorWarningID:= E_AlarmCategory.LifterStation2Device + 1, 
//	sDeviceID:= 'Lifter Station 2',
//	iSeverity:= 2, 
//	iNativeID:= 0, 
//	sNativeMessage:= 'Error Lifter Cylinder');

	
(*------------------------------------------------------------------------------------------------*)	
	
//Update alarm / warning list output to OPC
bST1ErrWarDataChange := iST1ErrWarDataChange <> Output.Station.Station1.ErrorWarning.DataChange;
iST1ErrWarDataChange := Output.Station.Station1.ErrorWarning.DataChange;
bST2ErrWarDataChange := iST2ErrWarDataChange <> Output.Station.Station2.ErrorWarning.DataChange;
iST2ErrWarDataChange := Output.Station.Station2.ErrorWarning.DataChange;
bTCErrWarDataChange := iTCErrWarDataChange <> fbTrack.stErrorWarning.DataChange;
iTCErrWarDataChange := fbTrack.stErrorWarning.DataChange;

IF bST1ErrWarDataChange OR bTCErrWarDataChange OR bCellDataChange THEN
	//Clear alarm list
	M_ErrorWarningClear();

	//Add alarm/warnings for Cell
	M_ErrorWarningAdd(arInErrorWarningList:= arErrorWarningDataCell, sLocationID:= 'C000004');
	
	//Add alarm/warnings for Station 1
	M_ErrorWarningAdd(arInErrorWarningList:= Output.Station.Station1.ErrorWarning.ErrorWarningData, sLocationID:= 'S000003');
	
	//Add alarm/warnings for Station 2
	M_ErrorWarningAdd(arInErrorWarningList:= Output.Station.Station2.ErrorWarning.ErrorWarningData, sLocationID:= 'S00000C');
	
	//Add alarm/warnings for Track Client
	M_ErrorWarningAdd(arInErrorWarningList:= fbTrack.stErrorWarning.ErrorWarningData, sLocationID:= 'TrackClient');
	
	stErrorWarning.DataChange := stErrorWarning.DataChange +1;
	//Output.Cell.ErrorWarning := stErrorWarning;
END_IF
END_METHOD

{attribute 'object_name' := 'M_Execute'}
METHOD M_Execute

IF (output.Station.Station1.ModeState.CurrentState = E_PML_State.Holding) THEN
	bHoldLocal := TRUE;
ELSIF (output.Station.Station1.ModeState.CurrentState = E_PML_State.Suspending) THEN
	bSuspendLocal := TRUE;
ELSIF (output.Station.Station1.ModeState.CurrentState <> E_PML_State.Execute) THEN
	// Exit execute state when all station(s) are not executing
	
	M_StateComplete();
END_IF
END_METHOD

{attribute 'object_name' := 'M_Held'}
METHOD M_Held
END_METHOD

{attribute 'object_name' := 'M_Holding'}
METHOD M_Holding

(*
// Check station(s) state
IF (fbBrushing.stOutput.stModeState.iCurrentState = E_PML_State.Held) THEN
	M_StateComplete();
END_IF
*)

// Do not wait for station state
//eCommand := E_PML_Command.Undefined;
M_StateComplete();
END_METHOD

{attribute 'object_name' := 'M_Idle'}
METHOD M_Idle
END_METHOD

METHOD PROTECTED M_Init : BOOL
VAR_INPUT
END_VAR

VAR
	SerialNumber: INT;
END_VAR
IF (NOT bInitDone) THEN
	// Set init done to TRUE. Set to false during init if needed
	bInitDone := TRUE;
	
	// test branch merge
	// test branch merge
	// test branch merge
	// test branch merge develop
	// test branch merge develop
	// test branch merge develop
	// test branch merge develop

// Track Client setup
	fbTrack.P_eCellType := E_CellType.Type_Inline;
	fbTrack.P_sCellID := 'C000004';
	fbTrack.P_sTrackserverURL := 'opc.tcp://10.38.190.121:4840';
	fbTrack.P_sTrackserverNetID := '10.38.190.121.1.1';
	fbTrack.P_nTrackserverPort := 851;
	//Next station on track
	fbTrack.P_sNextStationOnTrack := 'S000001';	// Cell 5
	// Paths
	
	// Station(s)
	bInitDone := bInitDone AND
	fbTrack.M_DefineStation(nStationNo := 1,
							sStationID := Input.Transport.Configuration.Stations[1].StationID,							//S000003
							nLoc1PathID := Input.Transport.Configuration.Stations[1].StationLocation1.Path,				//17
							rLoc1Position := Input.Transport.Configuration.Stations[1].StationLocation1.Position,		//1.000
							nLoc2PathID := 0, //Input.Transport.Configuration.Stations[1].StationLocation2.Path,
							rLoc2Position := 0, //Input.Transport.Configuration.Stations[1].StationLocation2.Position,
							nLocDecPathID := Input.Transport.Configuration.DecisionPointLocation.Path,					//17
							rLocDecPosition := Input.Transport.Configuration.DecisionPointLocation.Position,			//0.650
							nPreBufferSize := 0, //Input.Transport.Configuration.Stations[1].PreBufferSize,
							nPostBufferSize := 0); //Input.Transport.Configuration.Stations[1].PostBufferSize );
							
		fbTrack.M_DefineStation(nStationNo := 2,
							sStationID := Input.Transport.Configuration.Stations[2].StationID,							//S00000C
							nLoc1PathID := Input.Transport.Configuration.Stations[2].StationLocation1.Path,				//17
							rLoc1Position := Input.Transport.Configuration.Stations[2].StationLocation1.Position,		//1.850
							nLoc2PathID := 0, //Input.Transport.Configuration.Stations[2].StationLocation2.Path,
							rLoc2Position := 0, //Input.Transport.Configuration.Stations[2].StationLocation2.Position,
							nLocDecPathID := Input.Transport.Configuration.DecisionPointLocation.Path,					//17
							rLocDecPosition := Input.Transport.Configuration.DecisionPointLocation.Position,			//0.650
							nPreBufferSize := 0, //Input.Transport.Configuration.Stations[2].PreBufferSize,
							nPostBufferSize := 0); //Input.Transport.Configuration.Stations[2].PostBufferSize );
	
	// Cell information
	Output.Header.CellInformation.CellID := 'C000004';
	Output.Header.CellInformation.CellName := 'Cell 4';
	Output.Header.CellInformation.NumberOfStations := 2;
	Output.Header.MetaInformation.CellType := 'Inline';
	Output.Header.MetaInformation.InterfaceVersion := 0;
	Output.Header.MetaInformation.PLCVersion := nPLCVersion;
	Output.Header.MetaInformation.SerialNumber := sSerialIPC;
	
	// Station information
	Output.Header.CellInformation.StationInformation[1].NumberOfOperations := 1;
	Output.Header.CellInformation.StationInformation[1].StationID := 'S000003';
	Output.Header.CellInformation.StationInformation[1].StationName := 'HeatAndSteam In';
	Output.Station.Station1.CurrentConfiguration.OP11600.ToolCapacity := 0;
	Output.Station.Station1.CurrentConfiguration.OP11600.MaterialCapacity := 0;
	
	Output.Header.CellInformation.StationInformation[2].NumberOfOperations := 0;
	Output.Header.CellInformation.StationInformation[2].StationID := 'S00000C';
	Output.Header.CellInformation.StationInformation[2].StationName := 'HeatAndSteam Out';
//	Output.Station.Station2.CurrentConfiguration.OP11601.ToolCapacity := 0;
//	Output.Station.Station2.CurrentConfiguration.OP11601.MaterialCapacity := 0;

	
	// Operation information
	Output.Header.CellInformation.StationInformation[1].OperationInformation[1].OperationID := 'OP11600';
	Output.Header.CellInformation.StationInformation[1].OperationInformation[1].OperationName := 'HeatAndSteam Step 1';
	
	// Transport information
	Output.Header.CellInformation.TransportInformation.TransportName := 'C000004';
	Output.Header.CellInformation.TransportInformation.TransportType := 'Inline';
	
	// Components
	
	//Specify Sustainability data
	Output.Cell.SustainabilityData.Energy[1] := F_NewDeviceDataX(	'HS', 						'Heat and Steam', 
																	E_AlarmCategory.OP11600 +0, 	'Instant Power', 				E_Units._KW);
END_IF
END_METHOD

METHOD PROTECTED M_OEEHandling
VAR_INPUT
END_VAR
VAR
	bChanged			: BOOL;
END_VAR
// Call base FB method
SUPER^.M_OEEHandling();


// Product counters
IF ( stOEE.ProcessedProduct <> (Output.Station.Station1.OEE.ProcessedProduct) ) THEN
	stOEE.ProcessedProduct := Output.Station.Station1.OEE.ProcessedProduct;
	bChanged := TRUE;
END_IF
IF ( stOEE.GoodProduct <> (Output.Station.Station1.OEE.GoodProduct) ) THEN
	stOEE.GoodProduct := Output.Station.Station1.OEE.GoodProduct;
	bChanged := TRUE;
END_IF
IF ( stOEE.RejectedProduct <> (Output.Station.Station1.OEE.RejectedProduct) ) THEN
	stOEE.RejectedProduct := Output.Station.Station1.OEE.RejectedProduct;
	bChanged := TRUE;
END_IF

// Update Event ID!
// TODO!!!
stOEE.EventID;

// Increment DataChange to signal to LC that sometihng has changed
IF (bChanged) THEN
	// Update time for changes
	stOEE.DateTime := SYSTEMTIME_TO_DT(TIMESTR := fbGetTime.TIMESTR);
	
	stOEE.DataChange := stOEE.DataChange + 1;
END_IF
END_METHOD

{attribute 'object_name' := 'M_Resetting'}
METHOD M_Resetting
VAR
	bDone : BOOL;
END_VAR
// Track
fbTrack.bEnable := TRUE;

IF (fbTrack.bStarted AND fbTrack.bTrackInitDone AND fbTrack.bVehicleInitDone) OR bBypassTrack THEN
	eCommand := E_PML_Command.Undefined;
	M_StateComplete();
	bBypassTrack := FALSE;
END_IF
END_METHOD

{attribute 'object_name' := 'M_Starting'}
METHOD M_Starting
(*
// Check station(s)
IF (fbBrushing.stModeStateOut.CurrentState = E_PML_State.Execute) THEN
	bStartLocal := FALSE;
	M_StateComplete();
END_IF
*)

eCommand := E_PML_Command.Undefined;
M_StateComplete();
END_METHOD

{attribute 'object_name' := 'M_Stopped'}
METHOD M_Stopped
END_METHOD

{attribute 'object_name' := 'M_Stopping'}
METHOD M_Stopping
//eCommand := E_PML_Command.Undefined;
M_StateComplete();
END_METHOD

{attribute 'object_name' := 'M_Suspended'}
METHOD M_Suspended
END_METHOD

{attribute 'object_name' := 'M_Suspending'}
METHOD M_Suspending
//fbTrack.bSuspend := TRUE;

// Check station(s) state
//IF ( (output.Station.Station1.ModeState.CurrentState = E_PML_State.Suspended) AND fbTrack.bSuspended ) THEN
//	eCommand := E_PML_Command.Undefined;
	M_StateComplete();
//END_IF
END_METHOD

METHOD M_SustainabilityDataHandling
VAR_INPUT
END_VAR
Output.Cell.SustainabilityData.Energy[1].Value := Output.Station.Station1.OperationalData.OP11600.DeviceData[4].Value;
END_METHOD

{attribute 'object_name' := 'M_Undefined'}
METHOD M_Undefined
END_METHOD

{attribute 'object_name' := 'M_Unholding'}
METHOD M_Unholding

// Check station(s) state
IF ((output.Station.Station1.ModeState.CurrentState  <> E_PML_State.Held)) THEN
//	eCommand := E_PML_Command.Undefined;
	M_StateComplete();
END_IF
END_METHOD

{attribute 'object_name' := 'M_Unsuspending'}
METHOD M_Unsuspending
//eCommand := E_PML_Command.Undefined;
fbTrack.bSuspend := FALSE;
M_StateComplete();
(*
// Check station(s) state
IF (fbBrushing.stModeStateOut.CurrentState <> E_PML_State.Suspended) THEN
	M_StateComplete();
END_IF
*)
END_METHOD

METHOD M_VehicleOnStation : BOOL
VAR_INPUT
END_VAR
VAR
	bVehiclePresent			: BOOL;
	iCarrierIndex			: UINT;
	iCarrierID				: STRING;
	i						: UINT;
	j						: UINT;
	fPositionOut			: REAL;
	sTempString				: STRING(200);
END_VAR
VAR_OUTPUT
	iCarrierCount			: UINT;
END_VAR
//Carrier count
iCarrierCount := 0;
FOR i := 1 TO 10 DO
	IF (aVehiclesStationFIFO[i].sCarrierID = '') THEN
		EXIT;//End reached
	ELSE
		iCarrierCount := iCarrierCount + 1;
	END_IF 
END_FOR

CASE eSeq OF
	E_VehicleOnStation.Idle:
		IF fbTrack.bReadyStationIn[1] THEN
			stVehicleDataOnStation := fbTrack.P_stVehicleDataOnStation; //Read out vehicle data to temp
			eSeq := E_VehicleOnStation.VehicleAtStation;
			F_LogFile(CONCAT('Cell Vehicle On Station - New Vehicle station IN, Veh NO: ', TO_STRING(stVehicleDataOnStation.stVehicle.nVehicleID)));
		END_IF
		
	E_VehicleOnStation.VehicleAtStation:
		tonSeqTimer(IN := TRUE, PT := T#10S);
		IF output.Station.Station1.ModeState.CurrentState = E_PML_State.Starting (*AND NOT fbStationINHeatAndSteam.P_bSkipVehicle*) THEN
			tonSeqTimer(IN := FALSE);
			eSeq := E_VehicleOnStation.AddToFIFO;
			F_LogFile(CONCAT('Cell Vehicle On Station - Vehicle at station, Veh NO: ', TO_STRING(stVehicleDataOnStation.stVehicle.nVehicleID)));
//		ELSIF fbStationINHeatAndSteam.P_bSkipVehicle THEN
//			tonSeqTimer(IN := FALSE);
//			eSeq := E_VehicleOnStation.WaitStationStart;
//			F_LogFile(CONCAT('Cell Vehicle On Station - Vehicle at station SKIPPED, Veh NO: ', TO_STRING(stVehicleDataOnStation.stVehicle.nVehicleID)));
		END_IF
		
		// Check if vehicle is waiting for station start or skip
		IF (tonSeqTimer.Q) THEN
			// Force update of vehicle status to OPC/Line Controller
			tonSeqTimer(IN := FALSE);
			fbTrack.P_bForceVehicleUpdateOPC := TRUE;
		END_IF
		
	E_VehicleOnStation.AddToFIFO:
		
		FOR i := 1 TO 10 DO
			IF (aVehiclesStationFIFO[i].sCarrierID = '') THEN
				aVehiclesStationFIFO[i].sCarrierID := stVehicleDataOnStation.stVehicle.sCarrierID;
				aVehiclesStationFIFO[i].nVehicleNo := stVehicleDataOnStation.stVehicle.nVehicleID;
				aVehiclesStationFIFO[i].JobData := Output.Station.Station1.JobData.OP11600;
				aVehiclesStationFIFO[i].fVelocity := fbStationINHeatAndSteam.fVelocityCal;
				
				sTempString := CONCAT('Station FIFO - Carrier with ID: ', TO_STRING(aVehiclesStationFIFO[i].sCarrierID));
				sTempString := CONCAT(sTempString, ' added to FIFO, Vehicle no: ');
				sTempString := CONCAT(sTempString, TO_STRING(aVehiclesStationFIFO[i].nVehicleNo));
				sTempString := CONCAT(sTempString, ', Velocity: ');
				F_LogFIle(CONCAT(sTempString, TO_STRING(aVehiclesStationFIFO[i].fVelocity)));
				
				EXIT;
			END_IF
		END_FOR
		
		eSeq := E_VehicleOnStation.WaitStationStart;
		F_LogFile(CONCAT('Cell Vehicle On Station - Add FIFO, Veh NO: ', TO_STRING(stVehicleDataOnStation.stVehicle.nVehicleID)));
		
	E_VehicleOnStation.WaitStationStart:
	
		IF output.Station.Station1.ModeState.CurrentState = E_PML_State.Completing THEN
			//fbStationINHeatAndSteam.P_bSkipVehicle := FALSE;
			eSeq := E_VehicleOnStation.MoveVehicle;
			F_LogFile(CONCAT('Cell Vehicle On Station - Station completing, Veh NO: ', TO_STRING(stVehicleDataOnStation.stVehicle.nVehicleID)));
		END_IF
		
	E_VehicleOnStation.MoveVehicle:
		IF (fbStationINHeatAndSteam.P_bSkipVehicle) THEN
			// Set vehicle velocity to 1 if skipped!
			iRes := fbTrack.M_CallMoveVehicleToStationIn(	eInputType := E_MMVehicleInputType.eMMVehicleInputType_VehicleID, 
															sInput := UINT_TO_STRING(stVehicleDataOnStation.stVehicle.nVehicleID), 
															sStationID := fbTrack.aStations[2].sStationID,//'S00000C',
															eDirection := E_MMDirection.eMMDirection_Forward, 
															fVelocity := 1.0, 
															fAcceleration := 1	);
		ELSE
			iRes := fbTrack.M_CallMoveVehicleToStationIn(	eInputType := E_MMVehicleInputType.eMMVehicleInputType_VehicleID, 
															sInput := UINT_TO_STRING(stVehicleDataOnStation.stVehicle.nVehicleID), 
															sStationID := fbTrack.aStations[2].sStationID,//'S00000C',
															eDirection := E_MMDirection.eMMDirection_Forward, 
															fVelocity := fbStationINHeatAndSteam.fVelocityCal, 
															fAcceleration := 1	);
		END_IF

		IF (iRes = 2) THEN
			// Movement call OK
			fbTrack.P_bVehicleMovedFromSt1 := TRUE;
			eSeq := E_VehicleOnStation.VehicleLeftStation;
			
			sTempString := CONCAT('Cell Vehicle On Station - Vehicle No: ', TO_STRING(stVehicleDataOnStation.stVehicle.nVehicleID));
			sTempString := CONCAT(sTempString, ' Move OK towards station 2, with velocity: ');
			F_LogFIle(CONCAT(sTempString, TO_STRING(fbStationINHeatAndSteam.fVelocityCal)));
		ELSIF (iRes = 3) THEN
			// Movement call failed
			eSeq := E_VehicleOnStation.VehicleLeftStation;
			
			sTempString := CONCAT('Cell Vehicle On Station - Vehicle No: ', TO_STRING(stVehicleDataOnStation.stVehicle.nVehicleID));
			sTempString := CONCAT(sTempString, ' Move FAILED towards station 2, with velocity: ');
			F_LogFIle(CONCAT(sTempString, TO_STRING(fbStationINHeatAndSteam.fVelocityCal)));
		END_IF
	
	E_VehicleOnStation.VehicleLeftStation:
		eSeq := E_VehicleOnStation.Idle;
		
		F_LogFile(CONCAT('Cell Vehicle - Vehicle left station, Veh NO: ', TO_STRING(stVehicleDataOnStation.stVehicle.nVehicleID)));
END_CASE

//Remove from FIFO
IF fbTrack.P_iVehicleFifoOut > 0 THEN
	FOR i := 1 TO 9 DO
		IF aVehiclesStationFIFO[i].nVehicleNo = fbTrack.P_iVehicleFifoOut THEN
			sTempString := CONCAT('Cell VehicleOnStat: Vehicle#: ', TO_STRING(aVehiclesStationFIFO[1].nVehicleNo));
			fbTrack.M_VehicleToReadRemove(aVehiclesStationFIFO[1].nVehicleNo);
			sTempString := CONCAT(sTempString, ' Removed from FIFO place: ');
			F_LogFile(CONCAT(sTempString, TO_STRING(i)));
			
			aVehiclesStationFIFO[i] := aDummyVehicleStationData;
		END_IF
	END_FOR
	fbTrack.P_iVehicleFifoOut := 0;
END_IF
//IF fbTrack.P_bFifoOut THEN
	
//	IF (aVehiclesStationFIFO[1].sCarrierID <> '') THEN
//		sTempString := CONCAT('Station FIFO - FIFO out carrierID: ', TO_STRING(aVehiclesStationFIFO[1].sCarrierID));
//		fbTrack.M_VehicleToReadRemove(aVehiclesStationFIFO[1].nVehicleNo);
//		F_LogFIle(CONCAT(sTempString, ' Removed from FIFO'));
//	END_IF
		
//	aVehiclesStationFIFO[1].sCarrierID := '';
//	aVehiclesStationFIFO[1].fCalculatedTIA := 0.0;
//	aVehiclesStationFIFO[1].fVelocity := 0.0;
//	aVehiclesStationFIFO[1].nVehicleNo := 0;
//	fbTrack.P_bFifoOut := FALSE;
//END_IF


//Clean up FIFO
FOR i := 1 TO 9 DO
//	IF LEN(aVehiclesStationFIFO[i].sCarrierID) = 0 AND LEN(aVehiclesStationFIFO[i+1].sCarrierID) <> 0 THEN
	IF (aVehiclesStationFIFO[i].sCarrierID = '') AND (aVehiclesStationFIFO[i+1].sCarrierID <> '') THEN 
		aVehiclesStationFIFO[i] := aVehiclesStationFIFO[i+1]; // Move next item here
		aVehiclesStationFIFO[i+1] := aDummyVehicleStationData;
	END_IF
END_FOR	

//Update estimated time to reach station 2
tonVehicleDataRead(IN := TRUE, PT := T#1S);	// Read vehicle data every second
fPositionOut := Input.Transport.Configuration.Stations[2].StationLocation1.Position;
FOR i := 1 TO 10 DO
	IF (aVehiclesStationFIFO[i].sCarrierID = '') THEN
		EXIT;
	END_IF //End reached
	
	// Trig vehicle data reading
	IF (tonVehicleDataRead.Q) THEN
		fbTrack.M_VehicleToReadAdd(aVehiclesStationFIFO[i].nVehicleNo);
	END_IF
	
	FOR j := 1 TO 1000 DO
		IF (Output.Transport.Status.Carrier[i].CarrierID = '') THEN
			EXIT;
		END_IF //End reached
		
		IF (aVehiclesStationFIFO[i].sCarrierID = Output.Transport.Status.Carrier[j].CarrierID) THEN
			IF (aVehiclesStationFIFO[i].fVelocity > 0.001) THEN
				// Calculate remaining time for reaching station 2 location using remaining distance and commanded velocity
				aVehiclesStationFIFO[i].fCalculatedTIA := (Input.Transport.Configuration.Stations[2].StationLocation1.Position - Output.Transport.Status.Carrier[j].CurrentPosition) / aVehiclesStationFIFO[i].fVelocity;
			END_IF
		END_IF
	END_FOR
END_FOR
// Timer for reading vehicle data for vehicles in the FIFO buffer
IF (tonVehicleDataRead.Q) THEN
	tonVehicleDataRead(IN := FALSE);
END_IF

//Set empty out
M_VehicleOnStation := iCarrierCount = 0;

//Cyclic log FIFO timer
IF iCarrierCount > 0 THEN
	diFifoLogTimer := diFifoLogTimer + g_iPLCScan_MS;
	IF diFifoLogTimer > 10000 THEN
		FOR i := 1 TO iCarrierCount DO
			sTempString := CONCAT('Station FIFO - Status, Carrier ID: ', TO_STRING(aVehiclesStationFIFO[i].sCarrierID));
			sTempString := CONCAT(sTempString, ', Vehicle no: ');
			sTempString := CONCAT(sTempString, TO_STRING(aVehiclesStationFIFO[i].nVehicleNo));
			sTempString := CONCAT(sTempString, ', Velocity: ');
			sTempString := CONCAT(sTempString, TO_STRING(aVehiclesStationFIFO[i].fVelocity));
			sTempString := CONCAT(sTempString, ', TIA: ');
			F_LogFIle(CONCAT(sTempString, TO_STRING(aVehiclesStationFIFO[i].fCalculatedTIA)));
		END_FOR
		diFifoLogTimer := 0;
	END_IF
END_IF
END_METHOD

END_FUNCTION_BLOCK

// ---- POUs/MAIN.TcPOU
PROGRAM MAIN
VAR
	// OPC UA mapper for cell
	{attribute 'OPC.UA.DA':='1'}
	Bridge					: FB_OPC_Cell_Unit_4;

// Cell handling, PackML etc.
	fbUnit4					: FB_Cell_Unit_4;

// Log to file
	fbLogToFile				: FB_LogToFile;
	
//	LicenseState	AT %I*	: UINT;
	bInitDone 				: BOOL;
	
END_VAR

// test branch merge develop 
// test branch merge develop
// test branch merge develop


M_Init();

// Cell handling
fbUnit4(stModeStateIn := Bridge.Input.Cell.ModeState, 
		stModeStateOut := Bridge.Output.Cell.ModeState,
		stOEE := Bridge.Output.Cell.OEE,
		stErrorWarning := Bridge.Output.Cell.ErrorWarning,
		bResetEStop:= Bridge.P_bResetEStop,
		bLockDoor:= Bridge.P_bLockDoors, 
		bUnlockDoor:= Bridge.P_bUnlockDoors, 
		bCellLight:= Bridge.P_bCellLight,
		iHeartBeatFromMES:= Bridge.P_iHeartBeat,
		Input := Bridge.Input,		// Bridge Data Inputs
		Output := Bridge.Output, 	// Bridge Data Outputs
		bModeChangeInProcess=> 	);
		

// OPC handling
	// OPC handling
	Bridge.P_bEStop := fbUnit4.bEStopOK; 
	Bridge.P_bDoors := fbUnit4.bDoorsOK;
	Bridge.P_bCellLight := fbUnit4.bCellLightOn;
	Bridge.P_rPLCCPUTemp := fbUnit4.rCPUTemp;
	Bridge.P_rSafetyCPUTemp := fbUnit4.rSafetyTemp;
	Bridge.P_sPLCSerial := fbUnit4.sSerialIPC;
	Bridge.P_sPLCMBSerial := fbUnit4.sSerialMB;
	Bridge.P_bStationCommOK := NOT fbUnit4.bStationCommError;
	Bridge.P_iHeartBeat := fbUnit4.iHeartBeatToMES;
	Bridge.P_rOSCPULoad := fbUnit4.rCPULoad;
	Bridge.P_rPLCCPULoad := fbUnit4.rCPULoadPLC;
	Bridge.P_rCPUFrequency := fbUnit4.rCPUFrequency;
	Bridge();

//File logging
fbLocalTime(
	sNetID:= '', 
	bEnable:= TRUE, 
	dwCycle:= 5, 
	dwOpt:= 0, 
	tTimeout:=DEFAULT_ADS_TIMEOUT );	
	
fbLogToFile(Busy=> );

METHOD M_Init : BOOL
VAR_INPUT
END_VAR
// Init
IF (NOT bInitDone) THEN

	bInitDone := TRUE;
END_IF
END_METHOD

END_PROGRAM
